Fanuc KAREL source: KT00848.KL

PROGRAM KT00848
%NOLOCKGROUP
VAR
  Y1: ARRAY[2] OF BYTE
  Y2: ARRAY[2] OF BYTE
  OUT: INTEGER
BEGIN
  Y1[1] = 2
  Y2[1] = 3
  Y1[1] = 2
  Y2[1] = 3
  OUT = TAN(Y1[1])
END KT00848
